FUNCTION FC_NowAsDt : DT		// Returns the current time (=now) as 'DT'

FC_NowAsDt := FC_DateAndTimeToDt(iDateAndTime := FC_GetLocalDateAndTimeString());

END_FUNCTION

(* stored: Version 1.1.0.1, ProductVersion 3.1.4026.18
   POU FC_NowAsDt: Id {6b6fc9dd-7926-497d-ba0b-e895cf67f837}, SpecialFunc None *)
